FUNCTION Convert_ULINT_TO_TOD : BOOL
VAR_INPUT
	in : ULINT;
	out : REFERENCE TO TOD;
END_VAR
VAR
	converted : TOD;
END_VAR

converted := ULINT_TO_TOD(in);

IF (TOD_TO_ULINT(converted) <> in) THEN
	RETURN;
END_IF

out := converted;
Convert_ULINT_TO_TOD := TRUE;

END_FUNCTION

(* stored: Version 1.1.0.1, ProductVersion 3.1.4024.12
   POU Convert_ULINT_TO_TOD: Id {e106140b-57db-430f-bf1e-412299b31a60}, SpecialFunc None *)
